// TIA Portal project "Trabajo_asignatura" (V15)
// Consiste en realizar la programación de la siguiente secuencia de acciones usando el programa TIA Portal y un autómata S7-1200. Los elementos que nos encontraremos son un pulsador de marcha, un pulsador
// de paro, un LED de arranque máquina, un LED de apertura de puerta, la cinta transportadora A, la puerta y la cinta transportadora B.

(* hardware
DEVICE "S7-1200 station_1"  S7-1200 Station
   slot 0: "Rack_0"  S7-1200 Rack  Rack  V1.0
   slot 1: "PLC_1"  CPU 1214C AC/DC/Rly  6ES7 214-1BG40-0XB0  V4.2
*)

// ===== PLC "PLC_1"  CPU 1214C AC/DC/Rly =====

VAR_GLOBAL   // PLC tag table "Tabla de variables estándar"
   "Pulsador_Marcha" AT %I0.0 : Bool;
   "Pulsador_Paro" AT %I0.1 : Bool;
   "FC_Puerta_Abajo" AT %I0.2 : Bool;
   "FC_Puerta_Arriba" AT %I0.3 : Bool;
   "Contactor_Cinta_A" AT %Q0.0 : Bool;
   "Contactor_Subir_Puerta" AT %Q0.1 : Bool;
   "Contactor_Bajar_Puerta" AT %Q0.2 : Bool;
   "Contactor_Cinta_B" AT %Q0.3 : Bool;
   "LED_Arranque_Maquina" AT %Q0.4 : Bool;
   "LED_Apertura_Puerta" AT %Q0.5 : Bool;
END_VAR

DATA_BLOCK "AUX_FC1"   // DB1
TITLE = Auxiliares_FC1
{ S7_Optimized_Access := 'TRUE' }
AUTHOR : PabloGonzalezMartin
VERSION : 0.1
// Para gestionar el programa se podrá crear un DB (DB1 -> para marcas auxiliares del FC1, y DB2 -> para las marcas auxiliares del FC2) e ir declarando las bits auxiliares para la gestión del FC1 y FC2.
   VAR
      MF_Pulsador_M : Bool;   // Marca de flanco del pulsador de marcha
      MF_Pulsador_P : Bool;   // Marca de flanco del pulsador de paro
      Cinta_A : Bool;   // Movimiento de la cinta A
      Tiempo_arranque : Time := T#3s;   // Tiempo de arranque de la cinta A
      Valor_arranque : Time;   // Valor del tiempo de arranque de la cinta A
      Abrir_puerta : Bool;   // Apertura de la puerta
      Cerrar_puerta : Bool;   // Cerrado de la puerta
      Cinta_B : Bool;   // Movimiento de la cinta B
   END_VAR
BEGIN
END_DATA_BLOCK

DATA_BLOCK "AUX_FC2"   // DB2
TITLE = Auxiliares_FC2
{ S7_Optimized_Access := 'TRUE' }
AUTHOR : PabloGonzalezMartin
VERSION : 0.1
// Para gestionar el programa se podrá crear un DB (DB1 -> para marcas auxiliares del FC1, y DB2 -> para las marcas auxiliares del FC2) e ir declarando las bits auxiliares para la gestión del FC1 y FC2.
   VAR
      MF_Marcha : Bool;
      MF_Parada : Bool;
      LED_Verde : Bool;
      LED_Azul : Bool;
      Parapadeo_verde : Bool := false;
      Parpadeo_azul : Bool := false;
   END_VAR
BEGIN
END_DATA_BLOCK

// folder: System blocks/Program resources

DATA_BLOCK "IEC_Timer_0_DB"   // DB3
{ S7_Optimized_Access := 'TRUE' }
AUTHOR : Simatic
FAMILY : IEC
NAME : IEC_TMR
VERSION : 1.0
// stored: InstanceOfName IEC_TIMER
"IEC_TIMER"
BEGIN
END_DATA_BLOCK

DATA_BLOCK "IEC_Timer_0_DB_1"   // DB4
{ S7_Optimized_Access := 'TRUE' }
AUTHOR : Simatic
FAMILY : IEC
NAME : IEC_TMR
VERSION : 1.0
// stored: InstanceOfName IEC_TIMER
"IEC_TIMER"
BEGIN
END_DATA_BLOCK

DATA_BLOCK "IEC_Timer_0_DB_2"   // DB5
{ S7_Optimized_Access := 'TRUE' }
AUTHOR : Simatic
FAMILY : IEC
NAME : IEC_TMR
VERSION : 1.0
// stored: InstanceOfName IEC_TIMER
"IEC_TIMER"
BEGIN
END_DATA_BLOCK

DATA_BLOCK "IEC_Timer_0_DB_3"   // DB6
{ S7_Optimized_Access := 'TRUE' }
AUTHOR : Simatic
FAMILY : IEC
NAME : IEC_TMR
VERSION : 1.0
// stored: InstanceOfName IEC_TIMER
"IEC_TIMER"
BEGIN
END_DATA_BLOCK

DATA_BLOCK "IEC_Timer_0_DB_4"   // DB7
{ S7_Optimized_Access := 'TRUE' }
AUTHOR : Simatic
FAMILY : IEC
NAME : IEC_TMR
VERSION : 1.0
// stored: InstanceOfName IEC_TIMER
"IEC_TIMER"
BEGIN
END_DATA_BLOCK

// folder: (top level)

FUNCTION "Secuencia" : Void   // FC1, LAD
TITLE = FC_Secuencia
{ S7_Optimized_Access := 'TRUE' }
AUTHOR : PabloGonzalezMartin
VERSION : 0.1
// En este bloque se programará la secuencia de arranque y el paro de las cintas y la puerta activando las marcas auxiliares que en el FC de salidas activarán las salidas
   VAR_TEMP   // added for the SCL form of the ladder/FBD networks
      _w1 : Bool;
   END_VAR
BEGIN

REGION Network 1: Secuencia de arranque. Movimiento cinta A
   // Cuando se active el pulsador de marcha, en ese momento arrancará la cinta A. Se programará el pulsador como un flanco de bajada para evitar que en caso de avería por bloqueo del pulsador este se quede pulsado y produzca un error en el sistema.
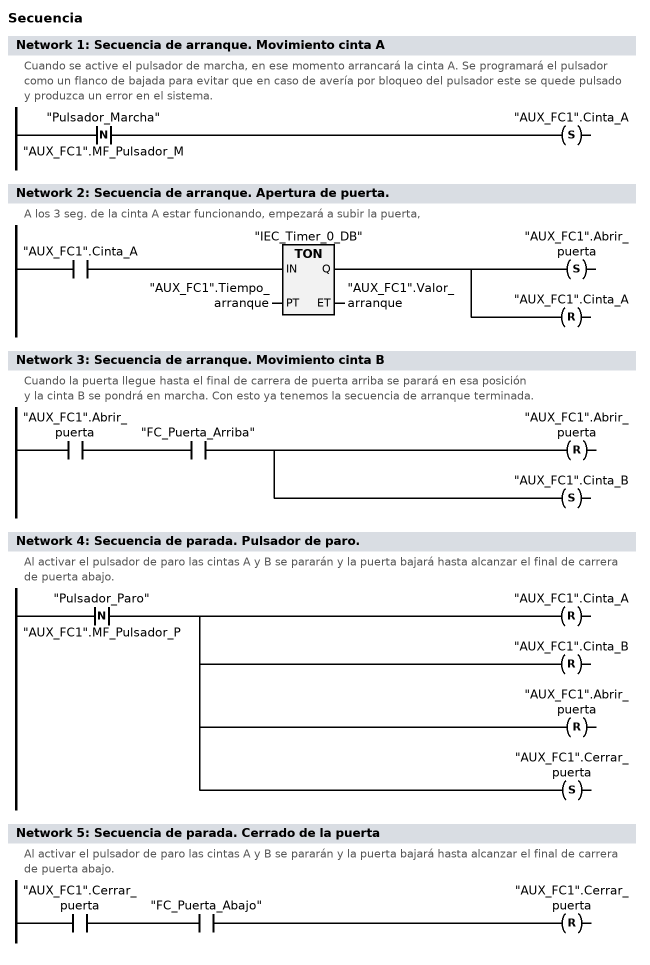
   RUNG wire#powerrail
      N_Contact(operand := "Pulsador_Marcha", bit := "AUX_FC1".MF_Pulsador_M)
      S_Coil( "AUX_FC1".Cinta_A )
   END_RUNG
   // the same network as SCL:
   #_w1 := NOT "Pulsador_Marcha" AND "AUX_FC1".MF_Pulsador_M;   // falling edge of "Pulsador_Marcha"
   "AUX_FC1".MF_Pulsador_M := "Pulsador_Marcha";
   IF #_w1 THEN "AUX_FC1".Cinta_A := TRUE; END_IF;
END_REGION

REGION Network 2: Secuencia de arranque. Apertura de puerta.
   // A los 3 seg. de la cinta A estar funcionando, empezará a subir la puerta,
   "IEC_Timer_0_DB".TON(IN := "AUX_FC1".Cinta_A,
                        PT := "AUX_FC1".Tiempo_arranque,
                        ET => "AUX_FC1".Valor_arranque);
   IF "IEC_Timer_0_DB".Q THEN
       "AUX_FC1".Abrir_puerta := TRUE;
       "AUX_FC1".Cinta_A := FALSE;
   END_IF;
END_REGION

REGION Network 3: Secuencia de arranque. Movimiento cinta B
   // Cuando la puerta llegue hasta el final de carrera de puerta arriba se parará en esa posición
   // y la cinta B se pondrá en marcha. Con esto ya tenemos la secuencia de arranque terminada.
   RUNG wire#powerrail
      Contact( "AUX_FC1".Abrir_puerta )
      Contact( "FC_Puerta_Arriba" )
      wire#w1
      R_Coil( "AUX_FC1".Abrir_puerta )
   END_RUNG
   RUNG wire#w1
      S_Coil( "AUX_FC1".Cinta_B )
   END_RUNG
   // the same network as SCL:
   #_w1 := "AUX_FC1".Abrir_puerta AND "FC_Puerta_Arriba";
   IF #_w1 THEN
       "AUX_FC1".Abrir_puerta := FALSE;
       "AUX_FC1".Cinta_B := TRUE;
   END_IF;
END_REGION

REGION Network 4: Secuencia de parada. Pulsador de paro.
   // Al activar el pulsador de paro las cintas A y B se pararán y la puerta bajará hasta alcanzar el final de carrera de puerta abajo.
   RUNG wire#powerrail
      N_Contact(operand := "Pulsador_Paro", bit := "AUX_FC1".MF_Pulsador_P)
      wire#w1
      R_Coil( "AUX_FC1".Cinta_A )
   END_RUNG
   RUNG wire#w1
      R_Coil( "AUX_FC1".Cinta_B )
   END_RUNG
   RUNG wire#w1
      R_Coil( "AUX_FC1".Abrir_puerta )
   END_RUNG
   RUNG wire#w1
      S_Coil( "AUX_FC1".Cerrar_puerta )
   END_RUNG
   // the same network as SCL:
   #_w1 := NOT "Pulsador_Paro" AND "AUX_FC1".MF_Pulsador_P;   // falling edge of "Pulsador_Paro"
   "AUX_FC1".MF_Pulsador_P := "Pulsador_Paro";
   IF #_w1 THEN
       "AUX_FC1".Cinta_A := FALSE;
       "AUX_FC1".Cinta_B := FALSE;
       "AUX_FC1".Abrir_puerta := FALSE;
       "AUX_FC1".Cerrar_puerta := TRUE;
   END_IF;
END_REGION

REGION Network 5: Secuencia de parada. Cerrado de la puerta
   // Al activar el pulsador de paro las cintas A y B se pararán y la puerta bajará hasta alcanzar el final de carrera de puerta abajo.
   RUNG wire#powerrail
      Contact( "AUX_FC1".Cerrar_puerta )
      Contact( "FC_Puerta_Abajo" )
      R_Coil( "AUX_FC1".Cerrar_puerta )
   END_RUNG
   // the same network as SCL:
   IF "AUX_FC1".Cerrar_puerta AND "FC_Puerta_Abajo" THEN "AUX_FC1".Cerrar_puerta := FALSE; END_IF;
END_REGION
END_FUNCTION

FUNCTION "LED" : Void   // FC2, LAD
TITLE = FC_LED
{ S7_Optimized_Access := 'TRUE' }
AUTHOR : PabloGonzalezMartin
VERSION : 0.1
// Se programará la gestión de los LED, dicha gestión activará las marcas correspondientes a cada LED.
   VAR_TEMP   // added for the SCL form of the ladder/FBD networks
      _w1 : Bool;
   END_VAR
BEGIN

REGION Network 1: Secuencia de arranque.
   // Cuando se active el pulsador de marcha, en ese momento comenzará a parpadear a una frecuencia de 2 Hz la luz verde.
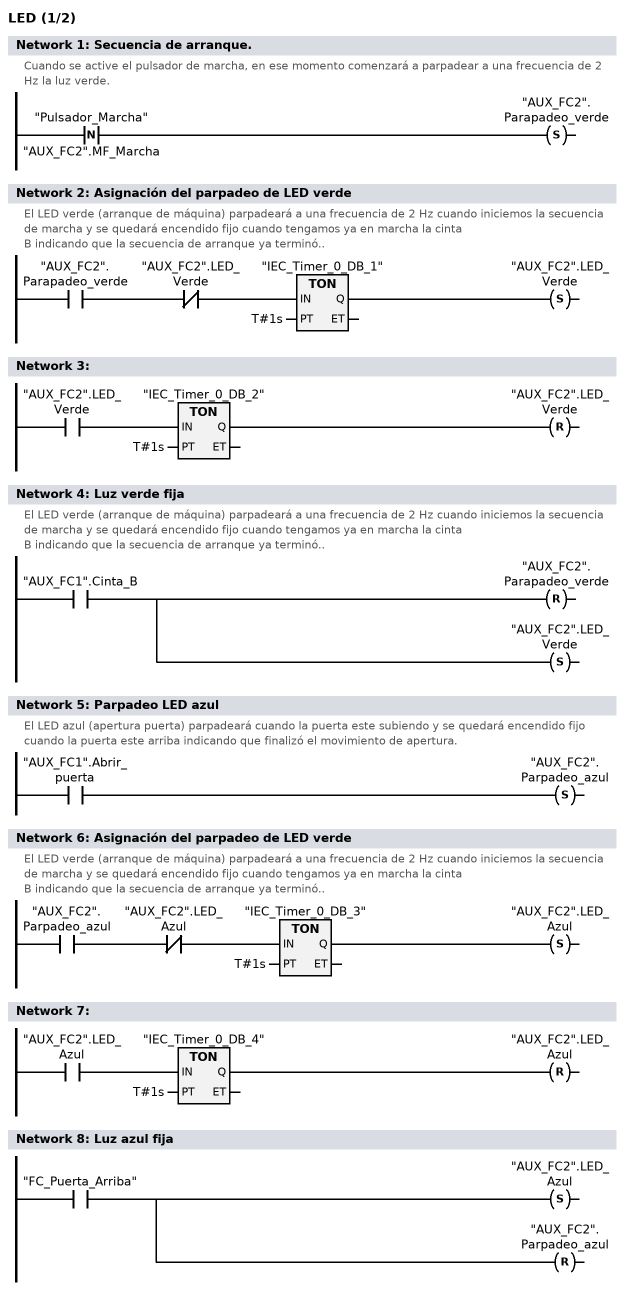
   RUNG wire#powerrail
      N_Contact(operand := "Pulsador_Marcha", bit := "AUX_FC2".MF_Marcha)
      S_Coil( "AUX_FC2".Parapadeo_verde )
   END_RUNG
   // the same network as SCL:
   #_w1 := NOT "Pulsador_Marcha" AND "AUX_FC2".MF_Marcha;   // falling edge of "Pulsador_Marcha"
   "AUX_FC2".MF_Marcha := "Pulsador_Marcha";
   IF #_w1 THEN "AUX_FC2".Parapadeo_verde := TRUE; END_IF;
END_REGION

REGION Network 2: Asignación del parpadeo de LED verde
   // El LED verde (arranque de máquina) parpadeará a una frecuencia de 2 Hz cuando iniciemos la secuencia de marcha y se quedará encendido fijo cuando tengamos ya en marcha la cinta
   // B indicando que la secuencia de arranque ya terminó..
   "IEC_Timer_0_DB_1".TON(IN := "AUX_FC2".Parapadeo_verde AND NOT "AUX_FC2".LED_Verde, PT := T#1s);
   IF "IEC_Timer_0_DB_1".Q THEN "AUX_FC2".LED_Verde := TRUE; END_IF;
END_REGION

REGION Network 3
   "IEC_Timer_0_DB_2".TON(IN := "AUX_FC2".LED_Verde, PT := T#1s);
   IF "IEC_Timer_0_DB_2".Q THEN "AUX_FC2".LED_Verde := FALSE; END_IF;
END_REGION

REGION Network 4: Luz verde fija
   // El LED verde (arranque de máquina) parpadeará a una frecuencia de 2 Hz cuando iniciemos la secuencia de marcha y se quedará encendido fijo cuando tengamos ya en marcha la cinta
   // B indicando que la secuencia de arranque ya terminó..
   RUNG wire#powerrail
      Contact( "AUX_FC1".Cinta_B )
      wire#w1
      R_Coil( "AUX_FC2".Parapadeo_verde )
   END_RUNG
   RUNG wire#w1
      S_Coil( "AUX_FC2".LED_Verde )
   END_RUNG
   // the same network as SCL:
   IF "AUX_FC1".Cinta_B THEN
       "AUX_FC2".Parapadeo_verde := FALSE;
       "AUX_FC2".LED_Verde := TRUE;
   END_IF;
END_REGION

REGION Network 5: Parpadeo LED azul
   // El LED azul (apertura puerta) parpadeará cuando la puerta este subiendo y se quedará encendido fijo cuando la puerta este arriba indicando que finalizó el movimiento de apertura.
   RUNG wire#powerrail
      Contact( "AUX_FC1".Abrir_puerta )
      S_Coil( "AUX_FC2".Parpadeo_azul )
   END_RUNG
   // the same network as SCL:
   IF "AUX_FC1".Abrir_puerta THEN "AUX_FC2".Parpadeo_azul := TRUE; END_IF;
END_REGION

REGION Network 6: Asignación del parpadeo de LED verde
   // El LED verde (arranque de máquina) parpadeará a una frecuencia de 2 Hz cuando iniciemos la secuencia de marcha y se quedará encendido fijo cuando tengamos ya en marcha la cinta
   // B indicando que la secuencia de arranque ya terminó..
   "IEC_Timer_0_DB_3".TON(IN := "AUX_FC2".Parpadeo_azul AND NOT "AUX_FC2".LED_Azul, PT := T#1s);
   IF "IEC_Timer_0_DB_3".Q THEN "AUX_FC2".LED_Azul := TRUE; END_IF;
END_REGION

REGION Network 7
   "IEC_Timer_0_DB_4".TON(IN := "AUX_FC2".LED_Azul, PT := T#1s);
   IF "IEC_Timer_0_DB_4".Q THEN "AUX_FC2".LED_Azul := FALSE; END_IF;
END_REGION

REGION Network 8: Luz azul fija
   RUNG wire#powerrail
      Contact( "FC_Puerta_Arriba" )
      wire#w1
      S_Coil( "AUX_FC2".LED_Azul )
   END_RUNG
   RUNG wire#w1
      R_Coil( "AUX_FC2".Parpadeo_azul )
   END_RUNG
   // the same network as SCL:
   IF "FC_Puerta_Arriba" THEN
       "AUX_FC2".LED_Azul := TRUE;
       "AUX_FC2".Parpadeo_azul := FALSE;
   END_IF;
END_REGION

REGION Network 9: Secuencia de parada. Pulsador de paro.
   // Al activar el pulsador de paro las cintas A y B se pararán y la puerta bajará hasta alcanzar el final de carrera de puerta abajo.
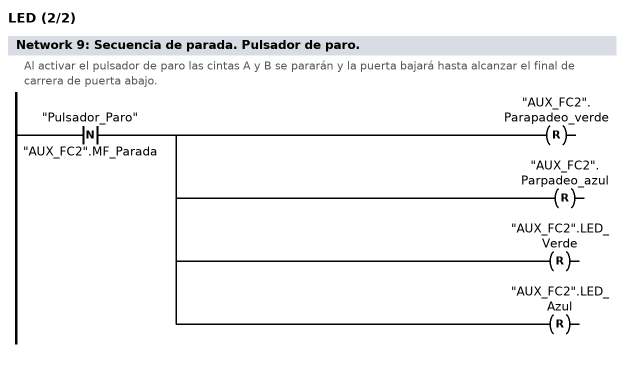
   RUNG wire#powerrail
      N_Contact(operand := "Pulsador_Paro", bit := "AUX_FC2".MF_Parada)
      wire#w1
      R_Coil( "AUX_FC2".Parapadeo_verde )
   END_RUNG
   RUNG wire#w1
      R_Coil( "AUX_FC2".Parpadeo_azul )
   END_RUNG
   RUNG wire#w1
      R_Coil( "AUX_FC2".LED_Verde )
   END_RUNG
   RUNG wire#w1
      R_Coil( "AUX_FC2".LED_Azul )
   END_RUNG
   // the same network as SCL:
   #_w1 := NOT "Pulsador_Paro" AND "AUX_FC2".MF_Parada;   // falling edge of "Pulsador_Paro"
   "AUX_FC2".MF_Parada := "Pulsador_Paro";
   IF #_w1 THEN
       "AUX_FC2".Parapadeo_verde := FALSE;
       "AUX_FC2".Parpadeo_azul := FALSE;
       "AUX_FC2".LED_Verde := FALSE;
       "AUX_FC2".LED_Azul := FALSE;
   END_IF;
END_REGION
END_FUNCTION

FUNCTION "Salidas" : Void   // FC3, LAD
TITLE = FC_Salidas
{ S7_Optimized_Access := 'TRUE' }
AUTHOR : PabloGonzalezMartin
VERSION : 0.1
// En este bloque se realizará la activación de las salidas por medio de las marcas auxiliares gestionadas en el FC1 de secuencia y el FC2 de LED, activando con cada una de ellas la salida correspondiente.
BEGIN

REGION Network 1: Asignacion de subir puerta
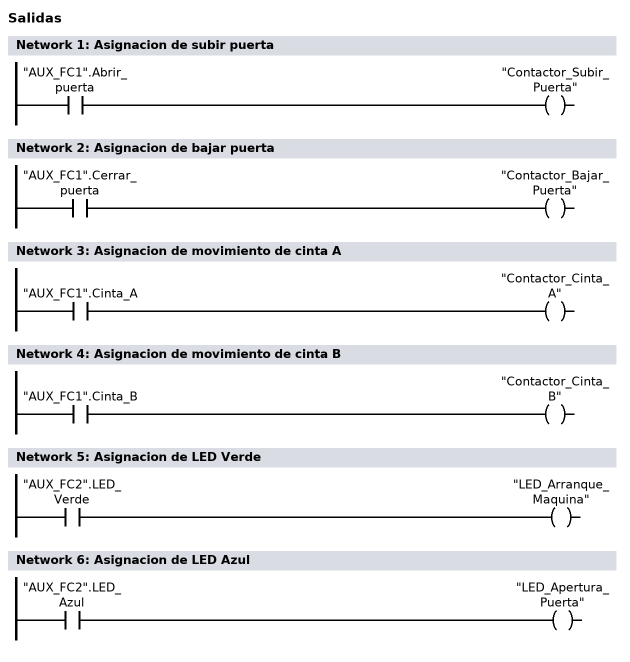
   RUNG wire#powerrail
      Contact( "AUX_FC1".Abrir_puerta )
      Coil( "Contactor_Subir_Puerta" )
   END_RUNG
   // the same network as SCL:
   "Contactor_Subir_Puerta" := "AUX_FC1".Abrir_puerta;
END_REGION

REGION Network 2: Asignacion de bajar puerta
   RUNG wire#powerrail
      Contact( "AUX_FC1".Cerrar_puerta )
      Coil( "Contactor_Bajar_Puerta" )
   END_RUNG
   // the same network as SCL:
   "Contactor_Bajar_Puerta" := "AUX_FC1".Cerrar_puerta;
END_REGION

REGION Network 3: Asignacion de movimiento de cinta A
   RUNG wire#powerrail
      Contact( "AUX_FC1".Cinta_A )
      Coil( "Contactor_Cinta_A" )
   END_RUNG
   // the same network as SCL:
   "Contactor_Cinta_A" := "AUX_FC1".Cinta_A;
END_REGION

REGION Network 4: Asignacion de movimiento de cinta B
   RUNG wire#powerrail
      Contact( "AUX_FC1".Cinta_B )
      Coil( "Contactor_Cinta_B" )
   END_RUNG
   // the same network as SCL:
   "Contactor_Cinta_B" := "AUX_FC1".Cinta_B;
END_REGION

REGION Network 5: Asignacion de LED Verde
   RUNG wire#powerrail
      Contact( "AUX_FC2".LED_Verde )
      Coil( "LED_Arranque_Maquina" )
   END_RUNG
   // the same network as SCL:
   "LED_Arranque_Maquina" := "AUX_FC2".LED_Verde;
END_REGION

REGION Network 6: Asignacion de LED Azul
   RUNG wire#powerrail
      Contact( "AUX_FC2".LED_Azul )
      Coil( "LED_Apertura_Puerta" )
   END_RUNG
   // the same network as SCL:
   "LED_Apertura_Puerta" := "AUX_FC2".LED_Azul;
END_REGION
END_FUNCTION

ORGANIZATION_BLOCK "Main"   // OB1, LAD, ProgramCycle
TITLE = "Main Program Sweep (Cycle)"
{ S7_Optimized_Access := 'TRUE' }
VERSION : 0.1
// : Únicamente se programará las llamadas a las bloques FC de secuencia, de LED y de salidas
   VAR_INPUT
      Initial_Call : Bool;   // Initial call of this OB
      Remanence : Bool;   // =True, if remanent data are available
   END_VAR
BEGIN

REGION Network 1: Llamada a la funcion de secuencia del programa
   // En este bloque se programará la secuencia de arranque y el paro de las cintas y la puerta activando las marcas auxiliares que en el FC de salidas activarán las salidas.
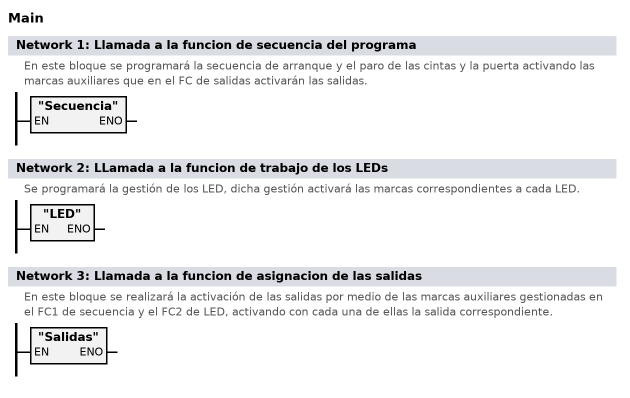
   RUNG wire#powerrail
      "Secuencia"()
   END_RUNG
   // the same network as SCL:
   "Secuencia"();
END_REGION

REGION Network 2: LLamada a la funcion de trabajo de los LEDs
   // Se programará la gestión de los LED, dicha gestión activará las marcas correspondientes a cada LED.
   RUNG wire#powerrail
      "LED"()
   END_RUNG
   // the same network as SCL:
   "LED"();
END_REGION

REGION Network 3: Llamada a la funcion de asignacion de las salidas
   // En este bloque se realizará la activación de las salidas por medio de las marcas auxiliares gestionadas en el FC1 de secuencia y el FC2 de LED, activando con cada una de ellas la salida correspondiente.
   RUNG wire#powerrail
      "Salidas"()
   END_RUNG
   // the same network as SCL:
   "Salidas"();
END_REGION
END_ORGANIZATION_BLOCK